// SIMATIC STEP 7 (V5.x) project TemperaturControl
// CPU: CPU315-2 DP(1)
// station: P_ADR_BUS
// station: Hardware
// station: SIMATIC 300 Station
// station: P_ADR_BUS
// station: Configuration
// program: S7 Program(1)

SYMBOL_TABLE
"Control"	DB 1	DB 1
"USEND"	FB 8	FB 8	// Uncoordinated Sending of Data
"CONT_C"	FB 41	FB 41	// Continuous Control
"CONT_S"	FB 42	FB 42	// Step Control
"TCONT_CP"	FB 58	FB 58	// temperature PID controller with pulse generator and self-tuning
"TCONT_S"	FB 59	FB 59	// temperature PID step controller
"HandMode"	FC 4	FC 4
"PUlSE"	FC 5	FC 5
"TIM_S5TI"	FC 40	FC 40	// IEC Time to S5 Time
"Fixed Number - Flt Pnt"	FC 61	FC 61	// Fixed number to floating point number
"SCALE"	FC 105	FC 105	// Scaling Values
"UpLimit"	I 0.2	BOOL
"leftLimit"	I 0.4	BOOL
"Up"	I 0.5	BOOL
"State"	M 1.0	BOOL
"OK"	M 55.0	BOOL
"alarmvar"	MW 10	WORD
"Sum"	MW 130	WORD
"Cycle Execution"	OB 1	OB 1
"CYC_INT5"	OB 35	OB 35	// Cyclic Interrupt 5
"HW_INT0"	OB 40	OB 40	// Hardware Interrupt 0
"DOWNWARD"	Q 4.0	BOOL
"GRASP"	Q 4.1	BOOL
"UPWARD"	Q 4.2	BOOL
"RIGHTWARD"	Q 4.3	BOOL
"LEFTWARD"	Q 4.4	BOOL
"BLKMOV"	SFC 20	SFC 20	// Copy Variables
"RDSYSST"	SFC 51	SFC 51	// Read a System Status List or Partial List
"WR_REC"	SFC 58	SFC 58	// Write Data Record
"RD_REC"	SFC 59	SFC 59	// Read a Data Record
"VAT_1"	VAT 1	
"VAT_2"	VAT 2	
END_SYMBOL_TABLE

FUNCTION_BLOCK FB 1
VERSION : 0.1
VAR_INPUT
  start : BOOL ;
  TON : TIMER ;
END_VAR
VAR_OUTPUT
  out : BOOL ;
END_VAR
VAR
  SetTime : S5TIME ;
END_VAR
BEGIN
NETWORK
TITLE =
      A     #start;
      L     #SetTime;
      T     LD 0;
      TAK;
      T     LD 4;
      L     #TON;
      T     LW 8;
      L     LD 4;
      L     LD 0;
      SD    T [LW 8];
      NOP   0;
      NOP   0;
      NOP   0;
      T     LD 0;
      TAK;
      T     LD 4;
      L     #TON;
      T     LW 8;
      L     LD 4;
      L     LD 0;
      A     T [LW 8];
      =     #out;
END_FUNCTION_BLOCK

// FB 8: know-how protected block, not included

FUNCTION_BLOCK FB 30
VERSION : 0.1
BEGIN
// (block stored without names or comments; labels and parameter names are numbered)
END_FUNCTION_BLOCK

// FB 58: know-how protected block, not included

FUNCTION FC 1 : VOID
VERSION : 0.1
VAR_INPUT
  PIW : INT ;
  HiLimit : REAL ;
  LowLimit : REAL ;
END_VAR
VAR_OUTPUT
  Temper : WORD ;
END_VAR
VAR_TEMP
  ret : WORD ;
  fcout : REAL ;
  truncout : DINT ;
  bipolar : BOOL ;
END_VAR
BEGIN
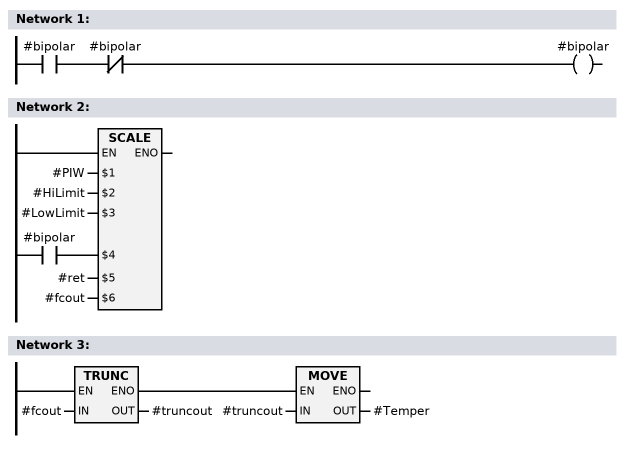
NETWORK
TITLE =
      A     #bipolar;
      AN    #bipolar;
      =     #bipolar;
NETWORK
TITLE =
      A     #bipolar;
      =     L 11.0;
      BLD   103;
      CALL  "SCALE" (
           $1                       := #PIW,
           $2                       := #HiLimit,
           $3                       := #LowLimit,
           $4                       := L 11.0,
           $5                       := #ret,
           $6                       := #fcout);
      NOP   0;
NETWORK
TITLE =
      A(;
      L     #fcout;
      TRUNC;
      T     #truncout;
      AN    OV;
      SAVE;
      CLR;
      A     BR;
      );
      JNB   _001;
      L     #truncout;
      T     #Temper;
_001: NOP   0;
END_FUNCTION

FUNCTION FC 2 : VOID
VERSION : 0.1
VAR_INPUT
  piw : INT ;
END_VAR
VAR_OUTPUT
  temper : WORD ;
END_VAR
BEGIN
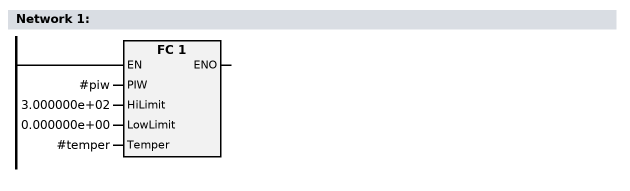
NETWORK
TITLE =
      CALL  FC 1 (
           PIW                      := #piw,
           HiLimit                  := 3.000000e+02,
           LowLimit                 := 0.000000e+00,
           Temper                   := #temper);
      NOP   0;
END_FUNCTION

FUNCTION FC 3 : VOID
VERSION : 0.1
VAR_IN_OUT
  inout1 : BOOL ;
END_VAR
BEGIN
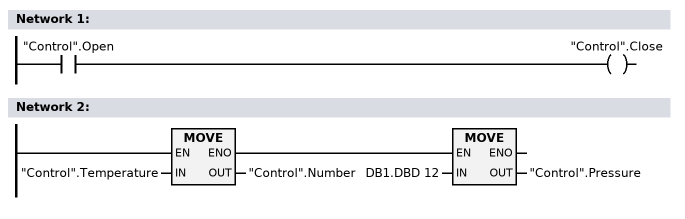
NETWORK
TITLE =
      A     "Control".Open;
      =     "Control".Close;
NETWORK
TITLE =
      A(;
      L     "Control".Temperature;
      T     "Control".Number;
      SET;
      SAVE;
      CLR;
      A     BR;
      );
      JNB   _001;
      L     DB1.DBD 12;
      T     "Control".Pressure;
_001: NOP   0;
NETWORK
TITLE =
END_FUNCTION

FUNCTION "HandMode" : VOID	// FC 4
VERSION : 0.1
BEGIN
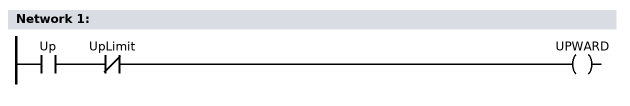
NETWORK
TITLE =
      A     "Up";
      AN    "UpLimit";
      =     "UPWARD";
END_FUNCTION

FUNCTION "PUlSE" : VOID	// FC 5
VERSION : 0.1
VAR_INPUT
  Enable : BOOL ;
  T : INT ;
END_VAR
VAR_OUTPUT
  Pulse_Out : BOOL ;
END_VAR
VAR_TEMP
  Dint_T : DINT ;
  S5T_T : S5TIME ;
  Time_T : TIME ;
  half_T : INT ;
END_VAR
BEGIN
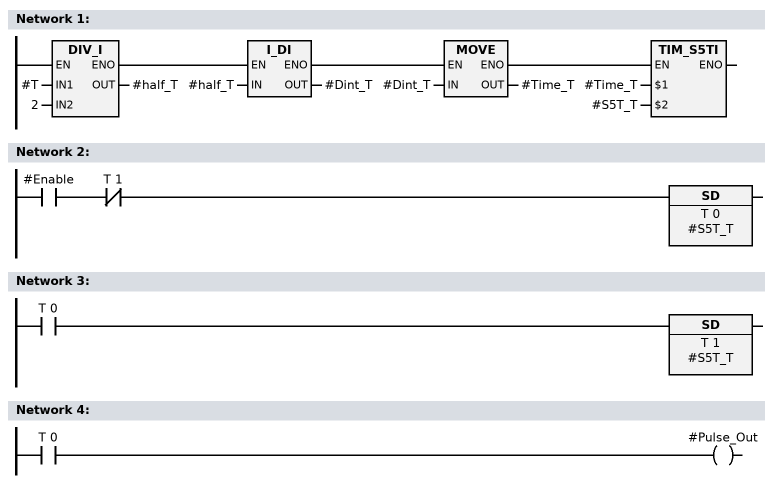
NETWORK
TITLE =
      A(;
      A(;
      A(;
      L     #T;
      L     2;
      /I;
      T     #half_T;
      AN    OV;
      SAVE;
      CLR;
      A     BR;
      );
      JNB   _001;
      L     #half_T;
      ITD;
      T     #Dint_T;
      SET;
      SAVE;
      CLR;
_001: A     BR;
      );
      JNB   _002;
      L     #Dint_T;
      T     #Time_T;
      SET;
      SAVE;
      CLR;
_002: A     BR;
      );
      JNB   _003;
      CALL  "TIM_S5TI" (
           $1                       := #Time_T,
           $2                       := #S5T_T);
_003: NOP   0;
NETWORK
TITLE =
      A     #Enable;
      AN    T 1;
      L     #S5T_T;
      SD    T 0;
NETWORK
TITLE =
      A     T 0;
      L     #S5T_T;
      SD    T 1;
NETWORK
TITLE =
      A     T 0;
      =     #Pulse_Out;
END_FUNCTION

FUNCTION FC 6 : VOID
VERSION : 0.1
BEGIN
NETWORK
TITLE =
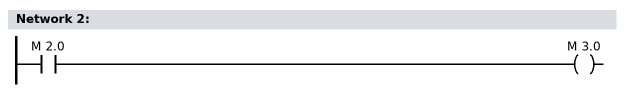
NETWORK
TITLE =
      A     M 2.0;
      =     M 3.0;
END_FUNCTION

// FC 40: know-how protected block, not included

// FC 61: know-how protected block, not included

// FC 105: know-how protected block, not included

DATA_BLOCK "Control"	// DB 1
VERSION : 0.1
  STRUCT
   Temperature : INT ;	//温度
   Pressure : REAL ;	//压力
   Open : BOOL ;	//打开
   Number : INT ;
   Close : BOOL ;	//关闭
   int3 : INT ;
  END_STRUCT ;	
BEGIN
END_DATA_BLOCK

DATA_BLOCK DB 2
VERSION : 0.1
  STRUCT
   alarm1 : STRING  [254 ] := 'limit reached';
  END_STRUCT ;	
BEGIN
   alarm1 := 'limit reached';
END_DATA_BLOCK

DATA_BLOCK DB 10
VERSION : 0.0
FB 1
BEGIN
END_DATA_BLOCK

DATA_BLOCK DB 58
AUTHOR : SIMATIC
FAMILY : CONTROL
VERSION : 0.0
"TCONT_CP"
BEGIN
END_DATA_BLOCK

DATA_BLOCK DB 100
VERSION : 0.0
FB 1
BEGIN
END_DATA_BLOCK

DATA_BLOCK DB 200
VERSION : 0.0
FB 1
BEGIN
END_DATA_BLOCK

ORGANIZATION_BLOCK "Cycle Execution"	// OB 1
TITLE = "Main Program Sweep (Cycle)"
VERSION : 0.1
VAR_TEMP
  OB1_EV_CLASS : BYTE ;	//Bits 0-3 = 1 (Coming event), Bits 4-7 = 1 (Event class 1)
  OB1_SCAN_1 : BYTE ;	//1 (Cold restart scan 1 of OB 1), 3 (Scan 2-n of OB 1)
  OB1_PRIORITY : BYTE ;	//Priority of OB Execution
  OB1_OB_NUMBR : BYTE ;	//1 (Organization block 1, OB1)
  OB1_RESERVED_1 : BYTE ;	//Reserved for system
  OB1_RESERVED_2 : BYTE ;	//Reserved for system
  OB1_PREV_CYCLE : INT ;	//Cycle time of previous OB1 scan (milliseconds)
  OB1_MIN_CYCLE : INT ;	//Minimum cycle time of OB1 (milliseconds)
  OB1_MAX_CYCLE : INT ;	//Maximum cycle time of OB1 (milliseconds)
  OB1_DATE_TIME : DATE_AND_TIME ;	//Date and time OB1 started
END_VAR
BEGIN
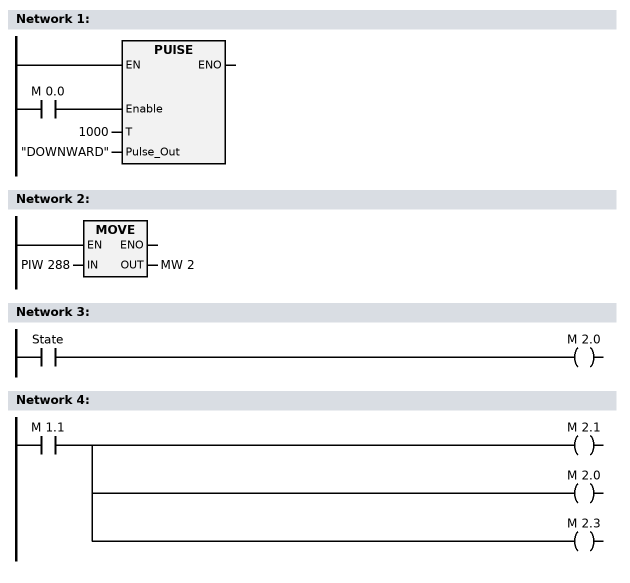
NETWORK
TITLE =
      A     M 0.0;
      =     L 20.0;
      BLD   103;
      CALL  "PUlSE" (
           Enable                   := L 20.0,
           T                        := 1000,
           Pulse_Out                := "DOWNWARD");
      NOP   0;
NETWORK
TITLE =
      L     PIW 288;
      T     MW 2;
      NOP   0;
NETWORK
TITLE =
      A     "State";
      =     M 2.0;
NETWORK
TITLE =
      A     M 1.1;
      =     M 2.1;
      =     M 2.0;
      =     M 2.3;
END_ORGANIZATION_BLOCK

ORGANIZATION_BLOCK "CYC_INT5"	// OB 35
TITLE = "Cyclic Interrupt"
VERSION : 0.1
VAR_TEMP
  OB35_EV_CLASS : BYTE ;	//Bits 0-3 = 1 (Coming event), Bits 4-7 = 1 (Event class 1)
  OB35_STRT_INF : BYTE ;	//16#36 (OB 35 has started)
  OB35_PRIORITY : BYTE ;	//Priority of OB Execution
  OB35_OB_NUMBR : BYTE ;	//35 (Organization block 35, OB35)
  OB35_RESERVED_1 : BYTE ;	//Reserved for system
  OB35_RESERVED_2 : BYTE ;	//Reserved for system
  OB35_PHASE_OFFSET : WORD ;	//Phase offset (msec)
  OB35_RESERVED_3 : INT ;	//Reserved for system
  OB35_EXC_FREQ : INT ;	//Frequency of execution (msec)
  OB35_DATE_TIME : DATE_AND_TIME ;	//Date and time OB35 started
END_VAR
BEGIN
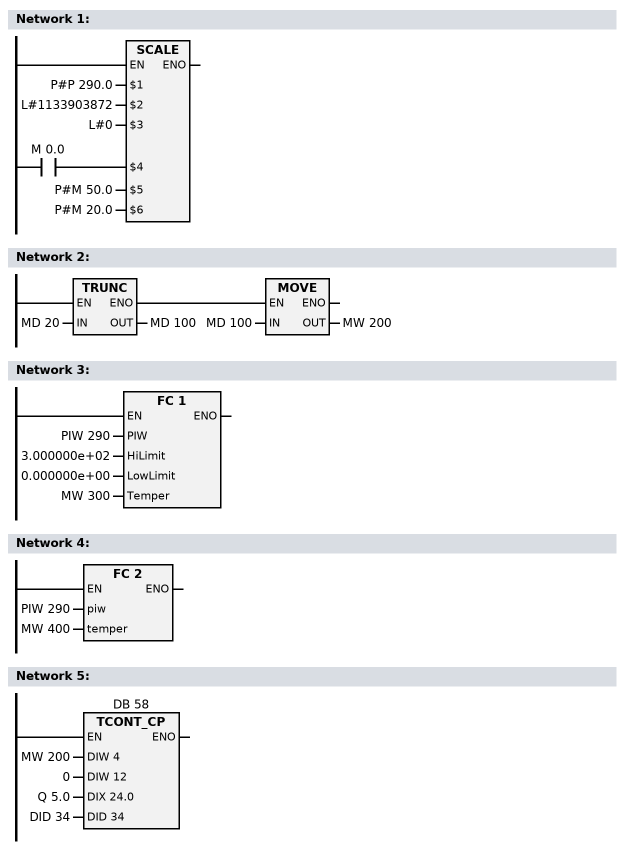
NETWORK
TITLE =
      A     M 0.0;
      =     L 20.0;
      BLD   103;
      CALL  "SCALE" (
           $1                       := P#P 290.0,
           $2                       := L#1133903872,
           $3                       := L#0,
           $4                       := L 20.0,
           $5                       := P#M 50.0,
           $6                       := P#M 20.0);
      NOP   0;
NETWORK
TITLE =
      A(;
      L     MD 20;
      TRUNC;
      T     MD 100;
      AN    OV;
      SAVE;
      CLR;
      A     BR;
      );
      JNB   _001;
      L     MD 100;
      T     MW 200;
_001: NOP   0;
NETWORK
TITLE =
      CALL  FC 1 (
           PIW                      := PIW 290,
           HiLimit                  := 3.000000e+02,
           LowLimit                 := 0.000000e+00,
           Temper                   := MW 300);
      NOP   0;
NETWORK
TITLE =
      CALL  FC 2 (
           piw                      := PIW 290,
           temper                   := MW 400);
      NOP   0;
NETWORK
TITLE =
      CALL  "TCONT_CP" , DB 58 (
           DIW 4                    := MW 200,
           DIW 12                   := 0,
           DIX 24.0                 := Q 5.0,
           DID 34                   := DID 34);
      NOP   0;
END_ORGANIZATION_BLOCK

ORGANIZATION_BLOCK "HW_INT0"	// OB 40
TITLE = "Hardware Interrupt"
VERSION : 0.1
VAR_TEMP
  OB40_EV_CLASS : BYTE ;	//Bits 0-3 = 1 (Coming event), Bits 4-7 = 1 (Event class 1)
  OB40_STRT_INF : BYTE ;	//16#41 (OB 40 has started)
  OB40_PRIORITY : BYTE ;	//Priority of OB Execution
  OB40_OB_NUMBR : BYTE ;	//40 (Organization block 40, OB40)
  OB40_RESERVED_1 : BYTE ;	//Reserved for system
  OB40_IO_FLAG : BYTE ;	//16#54 (input module), 16#55 (output module)
  OB40_MDL_ADDR : WORD ;	//Base address of module initiating interrupt
  OB40_POINT_ADDR : DWORD ;	//Interrupt status of the module
  OB40_DATE_TIME : DATE_AND_TIME ;	//Date and time OB40 started
END_VAR
BEGIN
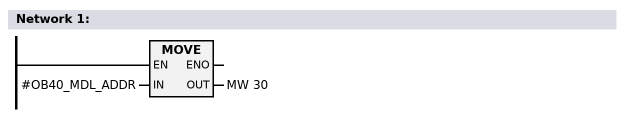
NETWORK
TITLE =
      L     #OB40_MDL_ADDR;
      T     MW 30;
      NOP   0;
END_ORGANIZATION_BLOCK
